FUNCTION_BLOCK fb_svControllers
VAR_INPUT
END_VAR
VAR_OUTPUT
END_VAR
VAR
END_VAR

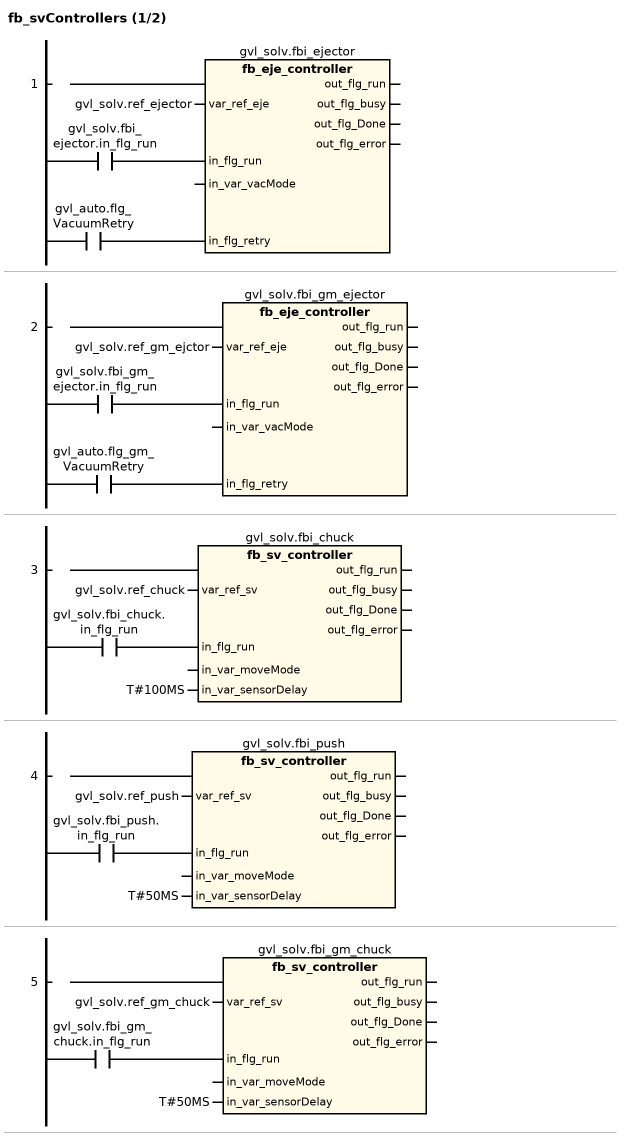
// NETWORK 1
gvl_solv.fbi_ejector(
    var_ref_eje := gvl_solv.ref_ejector,
    in_flg_run := gvl_solv.fbi_ejector.in_flg_run,
    in_flg_retry := gvl_auto.flg_VacuumRetry); // fb_eje_controller

// NETWORK 2
gvl_solv.fbi_gm_ejector(
    var_ref_eje := gvl_solv.ref_gm_ejctor,
    in_flg_run := gvl_solv.fbi_gm_ejector.in_flg_run,
    in_flg_retry := gvl_auto.flg_gm_VacuumRetry); // fb_eje_controller

// NETWORK 3
gvl_solv.fbi_chuck(
    var_ref_sv := gvl_solv.ref_chuck,
    in_flg_run := gvl_solv.fbi_chuck.in_flg_run,
    in_var_sensorDelay := T#100MS); // fb_sv_controller

// NETWORK 4
gvl_solv.fbi_push(
    var_ref_sv := gvl_solv.ref_push,
    in_flg_run := gvl_solv.fbi_push.in_flg_run,
    in_var_sensorDelay := T#50MS); // fb_sv_controller

// NETWORK 5
gvl_solv.fbi_gm_chuck(
    var_ref_sv := gvl_solv.ref_gm_chuck,
    in_flg_run := gvl_solv.fbi_gm_chuck.in_flg_run,
    in_var_sensorDelay := T#50MS); // fb_sv_controller

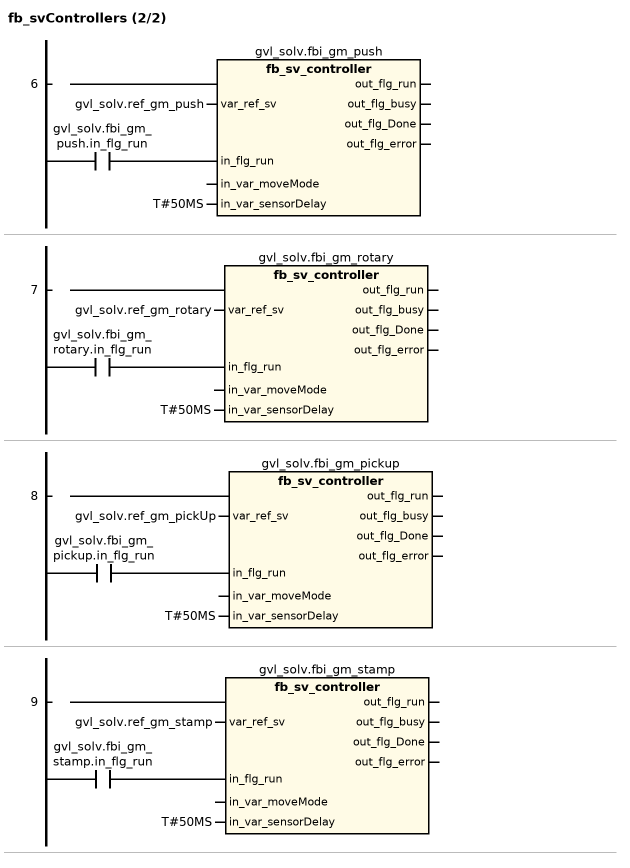
// NETWORK 6
gvl_solv.fbi_gm_push(
    var_ref_sv := gvl_solv.ref_gm_push,
    in_flg_run := gvl_solv.fbi_gm_push.in_flg_run,
    in_var_sensorDelay := T#50MS); // fb_sv_controller

// NETWORK 7
gvl_solv.fbi_gm_rotary(
    var_ref_sv := gvl_solv.ref_gm_rotary,
    in_flg_run := gvl_solv.fbi_gm_rotary.in_flg_run,
    in_var_sensorDelay := T#50MS); // fb_sv_controller

// NETWORK 8
gvl_solv.fbi_gm_pickup(
    var_ref_sv := gvl_solv.ref_gm_pickUp,
    in_flg_run := gvl_solv.fbi_gm_pickup.in_flg_run,
    in_var_sensorDelay := T#50MS); // fb_sv_controller

// NETWORK 9
gvl_solv.fbi_gm_stamp(
    var_ref_sv := gvl_solv.ref_gm_stamp,
    in_flg_run := gvl_solv.fbi_gm_stamp.in_flg_run,
    in_var_sensorDelay := T#50MS); // fb_sv_controller

END_FUNCTION_BLOCK

(* stored: Version 1.1.0.1, ProductVersion 3.1.4024.11
   POU fb_svControllers: Id {5944b19d-f503-4adf-b7b9-c88ea0e326aa}, SpecialFunc None *)
